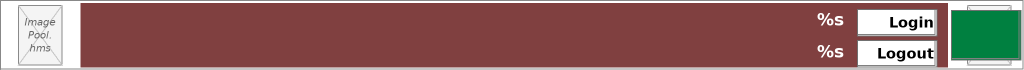
VISUALIZATION Header  // 1024x70
    Rectangle (77,0 947x70)
    Rectangle (535,39 312x25), "%s", text variable: visuelems.CurrentUserName
    Rectangle (948,0 79x70)
    Image (967,5 44x60), image: ImagePool.Logo
    Rectangle (0,72 1028x26), "MACHINE ERROR", invisible if: HMI_GVL.bMachineError
    Button (951,10 70x50), colour toggle: HMI_GVL.bMuteBuzzer, invisible if: HMI_GVL.bMachineError, image: VisuSymbols.Symbols.loudspeakerLoud
        toggle HMI_GVL.bMuteBuzzer
    Rectangle (1,1 79x70)
    Rectangle (0,72 1028x26), "REJECT FULL", invisible if: Status_GVL.RejectFull
    Image (18,5 44x60), image: ImagePool.hms
    Button (857,9 80x27), "Login", image: VisuSymbols.Symbols.User
        OnMouseDown: VisuUserMgmt Type=Login
    Rectangle (535,7 312x25), "%s", text variable: Status_GVL.strTimeEvent
    Button (857,40 80x27), "Logout", image: VisuSymbols.Symbols.User
        OnMouseDown: VisuUserMgmt Type=Logout
END_VISUALIZATION

(* stored: Version 1.1.0.1, ProductVersion 3.1.4024.12
   Visu Header: Id {2a7c5f77-be9e-4966-93c2-b6d28e297165} *)
